FUNCTION_BLOCK FB_ModbusComm
VAR_INPUT
END_VAR
VAR_OUTPUT
END_VAR
VAR
END_VAR

END_FUNCTION_BLOCK

(* stored: Version 1.1.0.1, ProductVersion 3.1.4024.13
   POU FB_ModbusComm: Id {1baef8da-7271-4b55-859d-971a63fa051c}, SpecialFunc None *)
